{attribute 'qualified_only'}
{attribute 'strict'}
TYPE MoveVelocitySequenceStep :
(
	Begin := 0,
  Exec,
  End
);
END_TYPE

(* stored: Version 1.1.0.1, ProductVersion 3.1.4024.11
   DUT MoveVelocitySequenceStep: Id {f7833724-70a1-46ae-b59e-81a6a611b1bb} *)
